// Function block searches all available tracking zones in range (Max 5 zones).
// This function block can be used to get how accurate a tu is positioned in a zone
FUNCTION_BLOCK FB_FindTrackingZones
(************************************************************************************** 
* 	Application 		: BoxControl Framework 
* 	Revision 			: $Revision: 408723 $ 
* 	Revision date 		: $Date: 2018-06-27 13:49:08 +0200 (Wed, 27 Jun 2018) $ 
* 	Last changed by 	: $Author: b7bolm $ 
* 	URL 				: $URL: http://almscdc.swisslog.com/repo/SWPD/Development/BoxControlFramework/21_Projects/BCF_2.0/trunk/BCF/BCF/JumpStart/20_Product/10_App/12_E_Functions/10_Lib/10_Conv/FB_FunctionList.TcPOU $ 
* ------------------------------------------------------------------------------------ 
* 	© Swisslog AG 
* 	Swisslog is not liable for any usage of this source code that is not agreed 
* 	on between Swisslog and the other party. The mandatory legal liability remains 
* 	unaffected. 
* ------------------------------------------------------------------------------------ 
* 	Revision History: 
* 
* 	VERSION 		DATE 			INITIALS 			DESCRIPTION 
* 	0.1 			30.11.2018 		mbo					First implementation
* 
**************************************************************************************)
VAR_INPUT
	Execute					: BOOL; // Rising edge triggers new search
	ObservationPosition		: UDINT; // Observation point [mm]
	Range					: UDINT; // Observation point +- Range defines area [mm]
	iWindowTracking			: I_WindowTracking; // Window tracking instance
END_VAR
VAR_OUTPUT
	TrackingZones			: ARRAY[1..MAX_ZONES] OF ST_TrackingZoneInfo; // Found tracking zones
	ZoneCounter 			: INT; // Found zones
	Error					: BOOL; // Configuration error
END_VAR
VAR
	Idx 					: INT; // Iterator
	TrackingZoneIndex		: UINT; // Found tracking zones
	fbTrig					: R_Trig; // Rising edge detection
	StartPosition			: UDINT; // Start search position
	EndPosition 			: UDINT; // End search position
	PositionDelta 			: DINT; // Delta zo zone begin
END_VAR
VAR CONSTANT
	MAX_ZONES				: INT := 5; // Max zones
END_VAR


fbTrig(CLK := Execute);

IF fbTrig.Q THEN
	// Check inputs
	IF iWindowTracking = 0 THEN
		Error := TRUE;
		RETURN;
	END_IF
	
	// Initialize
	Error := FALSE;
	StartPosition := ObservationPosition + Range;
	EndPosition := ObservationPosition - Range;
	ZoneCounter := 0;
	MEMSET(ADR(TrackingZones), 0, SIZEOF(TrackingZones));
	
	FOR Idx := 1 TO MAX_ZONES DO
		
		TrackingZoneIndex := iWindowTracking.M_GetFirstZoneIndex(
								mAbsoluteStartPosition := StartPosition,
								mAbsoluteEndPosition := EndPosition,
								mOnlyZonesWithTU := FALSE);
						
		IF TrackingZoneIndex > 0 THEN
			ZoneCounter := ZoneCounter + 1;
			
			IF ZoneCounter <= MAX_ZONES THEN
			
				PositionDelta := iWindowTracking.M_GetDistanceToZoneStart(ObservationPosition, TrackingZoneIndex);
				
				TrackingZones[ZoneCounter].ZoneIndex := TrackingZoneIndex;
				TrackingZones[ZoneCounter].PositionDelta := PositionDelta;
				TrackingZones[ZoneCounter].ZoneLength := iWindowTracking.P_ZoneTable[TrackingZoneIndex].ZoneLength;
			
				// Update next startposition to limit range
				StartPosition := EndPosition + 1;
			ELSE
				EXIT;
			END_IF
		// Otherwise no zone found, abort search
		ELSE
			EXIT;
		END_IF
	END_FOR
END_IF

END_FUNCTION_BLOCK

(* stored: Version 1.1.0.1, ProductVersion 3.1.4022.12
   POU FB_FindTrackingZones: Id {c067d9ed-dd14-4aaf-88b3-20537030cdfe}, SpecialFunc None *)
